// TIA Portal V17 export
// export: Created 2024-08-09T12:53:15.5373772Z, ExportSetting WithDefaults, DisplayName Totally Integrated Automation Portal, DisplayVersion V17 Update 7, DisplayName TIA Portal Openness, DisplayVersion V17 Update 7, DisplayName TIA Portal Version Control Interface, DisplayVersion V17, DisplayName STEP 7 Professional, DisplayVersion V17 Update 7, DisplayName STEP 7 Safety, DisplayVersion V17 Update 6, DisplayName WinCC Professional, DisplayVersion V17 Update 7
VAR_GLOBAL   // PLC tag table "CommunEns"
END_VAR
VAR_GLOBAL CONSTANT   // user constants
   ABANDONENS : USInt := 2;
   BTSUSPENS : USInt := 3;
   ARRET_NH : Char := 'N';
   ARRET_VID_NH : Char := 'H';
   ARRET_NB : Char := 'B';
END_VAR
